(* PLC project PlainProject, Unknown Unnamed 1 *)
(* stored: creationDateTime 2023-09-14T08:06:45, modificationDateTime 2023-09-14T08:09:26 *)

FUNCTION alpha : REAL
  VAR_INPUT  (* varGroup_44a5 *)
    q : REAL;  (* flow (m/3) *)
    Ts : REAL := 0.1;  (* sample time *)
    V : REAL := 1.0;  (* volume *)
  END_VAR

            alpha := q*Ts/V;
          
END_FUNCTION

FUNCTION density : REAL
  VAR_INPUT  (* varGroup_c33c *)
    temperature : REAL;  (* temperature *)
  END_VAR

            (* Specific density water *)

density := 1000.006621939
    + 0.00001626*temperature*temperature*temperature
    - 0.00602137*temperature*temperature
    + 0.02092985*temperature;
          
END_FUNCTION

FUNCTION heatCapacity : REAL
  VAR_INPUT  (* varGroup_1a63 *)
    temperature : REAL;
  END_VAR

            (* Specific heat capacity water *)
heatCapacity := 4201.7217960
   - 0.00013861*temperature*temperature*temperature
   + 0.03367866*temperature*temperature
   - 1.96518738*temperature;
          
END_FUNCTION

FUNCTION omega : REAL
  VAR_INPUT  (* varGroup_44a5 *)
    U : REAL;  (* thermal conductivity *)
    Ts : REAL := 0.1;  (* sample time *)
    V : REAL := 1.0;  (* Volume *)
    Temperature : REAL := 20.0;  (* temperature *)
  END_VAR

            omega := U*Ts/( density(Temperature)*heatCapacity(Temperature)*V );
          
END_FUNCTION

FUNCTION beta : REAL
  VAR_INPUT  (* varGroup_44a5 *)
    U : REAL;  (* thermal conductivity *)
    Ts : REAL := 0.1;  (* sample time *)
    V : REAL := 1.0;  (* Volume *)
    Temperature : REAL := 20.0;  (* temperature *)
    q : REAL;  (* flow *)
  END_VAR

            beta := 1.0 - omega(U:=U, Ts:=Ts, V:=V,Temperature:=Temperature) - alpha(q:=q, Ts:=Ts, V:=V);
          
END_FUNCTION

(* This is a heat exchanger FB *)
FUNCTION_BLOCK FB_heat_exchanger
  VAR CONSTANT  (* constants *)
    numberOfTanks : INT := 40;  (* discretization *)
  END_VAR
  VAR  (* varGroup_ffa7 *)
    index : INT;
    T1_k1 : ARRAY[0..40] OF REAL;  (* T1[k+1] Temp side 1, next timestep *)
    T2_k1 : ARRAY[0..40] OF REAL;  (* T2[k+1] Temp side 2, next timestep *)
    T1_k : ARRAY[0..40] OF REAL;  (* T1[k+1] Temp side 1, this timestep *)
    T2_k : ARRAY[0..40] OF REAL;  (* T2[k+1] Temp side 2, this timestep *)
    isInitialized : BOOL := false;
  END_VAR
  VAR  (* varGroup_2368 *)
    t1k1 : REAL;
    a1 : REAL;
    b1 : REAL;
    o1 : REAL;
    dens : REAL;
    heatCap : REAL;
  END_VAR
  VAR_INPUT  (* varGroup_fc5c *)
    Volume1 : REAL := 1.0;  (* total volume of side 1 [m3] *)
    Volume2 : REAL := 1.0;  (* total volume of side 2 [m3] *)
    Temperature1_In : REAL := 20.0;  (* Incoming T side 1 *)
    Temperature2_In : REAL := 20.0;  (* Incoming T side 2 *)
    q1 : REAL := 1.0;  (* Flow side 1 m3/s *)
    q2 : REAL := 1.0;  (* Flow side 2 m3/s *)
    Ts : REAL := 0.1;  (* sample time *)
    U : REAL;  (* thermal conductivity[W/K] *)
  END_VAR
  VAR_OUTPUT  (* varGroup_e821 *)
    Temperature1_Out : REAL;
    Temperature2_Out : REAL;
  END_VAR

            if NOT isInitialized then
    isInitialized := true;
    FOR index := 0 TO numberOfTanks DO
        T1_k[index] := Temperature2_In;
        T2_k[index] := Temperature2_In;
    END_FOR;
    dens := density(T1_k[0]);
    heatCap := heatCapacity(T1_k[0]);
    a1 := alpha(q:=q1, Ts:=Ts, V:=Volume1)*T1_k[0];
    b1 := beta(U:=U, Ts:=Ts, V:=Volume1, Temperature:=T1_k[1], q:=q1)*T1_k[1];
    o1 := omega(U:=U, Ts:=Ts, V:=Volume1, Temperature:=T1_k[1])*T2_k[40];
        
    t1k1 := a1+b1+o1;
END_IF;

T1_k[0] := Temperature1_In;
T2_k[0] := Temperature2_In;
FOR index := 1 TO numberOfTanks DO
    T1_k1[index] := alpha(q:=q1, Ts:=Ts, V:=Volume1)*T1_k[index-1]
        +beta(U:=U, Ts:=Ts, V:=Volume1, Temperature:=T1_k[index], q:=q1)*T1_k[index]
        +omega(U:=U, Ts:=Ts, V:=Volume1, Temperature:=T1_k[index])*T2_k[numberOfTanks-index+1];
    T2_k1[index] := alpha(q:=q2, Ts:=Ts, V:=Volume2)*T2_k[index-1]
        +beta(U:=U, Ts:=Ts, V:=Volume2, Temperature:=T2_k[index], q:=q2)*T2_k[index]
        +omega(U:=U, Ts:=Ts, V:=Volume2, Temperature:=T2_k[index])*T1_k[numberOfTanks-index+1];
END_FOR;

Temperature1_Out := T1_k[numberOfTanks];
Temperature2_Out := T2_k[numberOfTanks];

(* Move next step into current step *)
T1_k := T1_k1;
T2_k := T2_k1;

          
END_FUNCTION_BLOCK

PROGRAM program0
  VAR  (* Heat exchanger *)
    heatExhanger1 : FB_heat_exchanger;
    T1_in : REAL := 40.0;
    T2_in : REAL := 10.0;
    T1_out : REAL;
    T2_out : REAL;
    q1 : REAL := 140.0;
    q2 : REAL := 60.0;
    heatTransferNumber : REAL;
    heatTransferArea : REAL;
    volumeDiscretization : REAL;
    inletFlow_WarmSide : REAL;
  END_VAR
  VAR  (* controller *)
    Side2_controller : PID;
    PID_kp : REAL := 4.0;
    PID_tr : REAL := 100.0;
    PID_td : REAL := 0.0;
    PID_AUTO : BOOL;
    PID_sp : REAL := 30.0;
    valve_opening : REAL;
    PID_X0 : REAL := 12.5;
  END_VAR

            (*                  Heat Exchanger

side 1 In -->  |  =====>====>====>====>====> |  --> side 1 Out
               |                             |
               |                             |
side 2 Out <-- |  <====<====<====<====<====  |  <-- side 2 In

max inlet flow :
  side 1 140 m3/h
  side 2 60 m3/h

Play with the exchanger by changing the following values:
  T1_in,T2_in,q1,q2

*)

heatTransferArea := 37.0; (* m2 *)
heatTransferNumber := 4839.0; (* W/m2*K *)
volumeDiscretization := 40.0;

heatExhanger1(
  Volume1 := 0.0047,    (* total volume of side 1 [m3]*)
  Volume2 := 0.0038,    (* total volume of side 2 [m3]*)
  Temperature1_In := T1_in,    (* Incoming T side 1 [C] *)
  Temperature2_In := T2_in,    (* Incoming T side 2 [C] *)
  q1 := inletFlow_WarmSide/3600.0,    (* Flow side 1 [m3/s] *)
  q2 := q2/3600.0,    (* Flow side 2 [m3/s] *)
  Ts := 0.1,    (* sample time [s]*)
  U := heatTransferNumber*heatTransferArea/volumeDiscretization,    (* thermal conductivity [W/K] *)
  
  Temperature1_Out => T1_out,
  Temperature2_Out => T2_out
);

Side2_controller(
  (* Inputs *)
  AUTO := PID_AUTO,
  PV := T2_out,
  SP := PID_sp,
  KP := PID_kp,
  TR := PID_tr,
  TD := PID_td,
  X0 := PID_X0, (* start bias *)
  CYCLE := T#100ms
);

(* output limitation *)
if Side2_controller.XOUT < 0.0 then
  valve_opening := 100.0;
elsif Side2_controller.XOUT > 100.0 then  
  valve_opening := 0.0;
else 
  valve_opening := 100.0-Side2_controller.XOUT;
end_if;
inletFlow_WarmSide := q1*valve_opening/100.0;

(* fuzzy antiwindup *)
if Side2_controller.XOUT < 0.0 then
  PID_AUTO := false;
elsif Side2_controller.XOUT > 100.0 then
  PID_AUTO := false;
ELSE
  PID_AUTO := true;
END_IF;
          
END_PROGRAM

CONFIGURATION config
  RESOURCE resource1 ON PLC
    TASK task0(INTERVAL := T#100ms, PRIORITY := 0);
    PROGRAM instance0 WITH task0 : program0;
  END_RESOURCE
END_CONFIGURATION
